// TIA Portal V16 export
// export: Created 2021-10-04T12:51:10.0135951Z, ExportSetting WithDefaults, DisplayName Totally Integrated Automation Portal, DisplayVersion V16, DisplayName TIA Portal Version Control Interface, DisplayVersion V16, DisplayName TIA Portal Openness, DisplayVersion V16, DisplayName STEP 7 Professional, DisplayVersion V16, DisplayName STEP 7 Safety, DisplayVersion V16, DisplayName WinCC Advanced, DisplayVersion V16
FUNCTION_BLOCK "SmartTimer"   // FB1, LAD
{ S7_Optimized_Access := 'TRUE' }
VERSION : 0.1
// stored: AutoNumber true, IsIECCheckEnabled false, IsRetainMemResEnabled false, MemoryReserve 100, SetENOAutomatically false, UDAEnableTagReadback false
   VAR_INPUT
      "Time" : Time;
   END_VAR
   VAR_OUTPUT
      Q : Bool;
   END_VAR
   VAR
      IEC_Timer_0_Instance { S7_SetPoint := 'True'} : TON_TIME;
   END_VAR
BEGIN

REGION Network 1
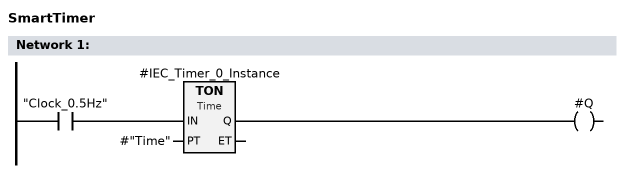
   RUNG wire#powerrail
      Contact( "Clock_0.5Hz" )
      { S7_Templates := "time_type := Time" } #IEC_Timer_0_Instance.TON(pt := #"Time", et =>)
      Coil( #Q )
   END_RUNG
   // the same network as SCL:
   #IEC_Timer_0_Instance(IN := "Clock_0.5Hz", PT := #"Time");   // TON
   #Q := #IEC_Timer_0_Instance.Q;
END_REGION
END_FUNCTION_BLOCK
